{attribute 'qualified_only'}
VAR_GLOBAL
	sModeDisplay : STRING;
	bGreenLed : BOOL;
	bRedLed : BOOL;
	fJoyStickSignal : REAL;
END_VAR

(* stored: Version 1.1.0.1, ProductVersion 3.1.4024.10
   GVL G_Output: Id {393b3012-cae2-45bd-a497-9c5c354eafb2} *)
